FUNCTION_BLOCK Cu00xTestPositions EXTENDS TcoDrivesBeckhoff.TcoSingleAxisPositionsRootContainer
VAR_INPUT
END_VAR
VAR_OUTPUT
END_VAR
VAR
	{attribute addProperty Name "<#Pick Position#>"}
	PickPosition:TcoDrivesBeckhoff.TcoSingleAxisMoveParam;
	{attribute addProperty Name "<#Place  Position#>"}
	PlacePosition:TcoDrivesBeckhoff.TcoSingleAxisMoveParam;
END_VAR

END_FUNCTION_BLOCK

(* stored: Version 1.1.0.1
   POU Cu00xTestPositions: Id {4fd6a69c-a695-462f-a5d8-c710bf5e640a}, SpecialFunc None *)
